(* Logix 5000 project; controller SEER_TEMPLATE vendor 1 type 14 code 54 rev 17.2; software revision 17.00 *)
// SEER_TEMPLATE

TASK MainTask (continuous, watchdog 500 ms) : MainProgram

MODULES
   Local : vendor 1 type 14 code 54 (ICP 0, rev 17.2)
END_MODULES

VAR_GLOBAL   (* controller tags *)
   F101x0 : REAL;   // SEER_IO_1 ANALOG COMM NULL REGISTER(S)
   F101x1 : REAL;   // SEER_IO_1 ANALOG COMM CYCLE TOTALIZER
   F101x2 : REAL;   // SEER_IO_1 ANALOG COMM JOB NUMBER
   F101x3 : REAL;   // SEER_IO_1 ANALOG COMM SCHEDULE NUMBER
   F101x4 : REAL;   // SEER_IO_1 ANALOG COMM OPERATOR ID
   N100x0 : INT;   // SEER_IO_0 DISCRETE COMM BINARY ELEMENTS INCLUDED
        .1   // SEER_IO_0 DISCRETE COMM CYCLE RESET COMMAND TRIGGER
        .2   // SEER_IO_0 DISCRETE COMM CYCLE RESET ONE SHOT
        .3   // SEER_IO_0 DISCRETE COMM MACHINE IS IN MAINTENANCE MODE
        .4   // SEER_IO_0 DISCRETE COMM CYCLE COUNT +1 ONE SHOT
        .5   // SEER_IO_0 DISCRETE COMM CYCLE COUNT +1 CYCLE DETECTED
        .6   // SEER_IO_0 DISCRETE COMM NO MACHINE ALARMS HAVE BEEN DETECTED
        .7   // SEER_IO_0 DISCRETE COMM NO MAJOR ALARMS HAVE BEEN DETECTED
        .8   // SEER_IO_0 DISCRETE COMM NO MINOR ALARMS HAVE BEEN DETECTED
        .9   // SEER_IO_0 DISCRETE COMM IDLE WITHOUT CYCLE DETECTED
        .11   // SEER_IO_0 DISCRETE COMM JOB '0' ONE SHOT
        .12   // SEER_IO_0 DISCRETE COMM JOB '0' ACTIVE NO JOB RUNNING
        .10   // SEER_IO_0 DISCRETE COMM ALWAYS FALSE INSTRUCTION (ALWAYS = 0)
   N100x1 : INT;   // SEER_IO_0 TEMPLATE TUTORIAL REGISTERS (REPLACE WITH YOUR BITS AND TAGS)
        .0   // SEER_IO_0 TEMPLATE TUTORIAL REPLACE WITH SOME LOGIC TO INDICATE PACKAGE TYPE "1"
        .1   // SEER_IO_0 TEMPLATE TUTORIAL REPLACE WITH SOME LOGIC TO INDICATE PACKAGE TYPE "2"
        .2   // SEER_IO_0 TEMPLATE TUTORIAL REPLACE WITH SOME LOGIC TO INDICATE PACKAGE TYPE "3"
        .3   // SEER_IO_0 TEMPLATE TUTORIAL REPLACE WITH SOME LOGIC TO INDICATE CUSTOM ALARM "1"
        .4   // SEER_IO_0 TEMPLATE TUTORIAL REPLACE WITH SOME LOGIC TO INDICATE CUSTOM ALARM "2"
        .5   // SEER_IO_0 TEMPLATE TUTORIAL REPLACE WITH SOME LOGIC TO INDICATE CUSTOM ALARM "3"
        .6   // SEER_IO_0 TEMPLATE TUTORIAL REPLACE WITH SOME LOGIC TO INDICATE CUSTOM ALARM "4"
        .7   // SEER_IO_0 TEMPLATE TUTORIAL REPLACE WITH SOME LOGIC TO INDICATE CUSTOM WARNING "1"
        .8   // SEER_IO_0 TEMPLATE TUTORIAL REPLACE WITH SOME LOGIC TO INDICATE CUSTOM WARNING "2"
        .9   // SEER_IO_0 TEMPLATE TUTORIAL REPLACE WITH SOME LOGIC TO INDICATE CUSTOM WARNING "3"
        .10   // SEER_IO_0 TEMPLATE TUTORIAL REPLACE WITH SOME LOGIC TO INDICATE THAT THE MACHINE HAS CYCLED 1 TIME
   N100x2 : INT;   // SEER_IO_0 DISCRETE COMM ALARM STATE
   N100x3 : INT;   // SEER_IO_0 DISCRETE COMM ALARM STATE PENDING
   N100x4 : INT;   // SEER_IO_0 DISCRETE COMM MACHINE STATE
   N100x5 : INT;   // SEER_IO_0 DISCRETE COMM CORRECTIVE ACTION
   N100x6 : INT;   // SEER_IO_0 DISCRETE COMM PACKAGES PER CYCLE
   N100x7 : INT;   // SEER_IO_0 DISCRETE COMM PACKAGE CLASS (TYPE)
   N100x8 : INT;   // SEER_IO_0 DISCRETE COMM MAJOR ALARM ID PENDING
   N100x9 : INT;   // SEER_IO_0 DISCRETE COMM MINOR ALARM ID PENDING
   T102x0 : TIMER := (PRE := 240000);   // SEER_IO_2 TIMERS IDLE TIME WITHOUT CYCLE DETECTED TIME BASE = 0.001 SEC
END_VAR

PROGRAM MainProgram   (* main routine MainRoutine *)

ROUTINE MainRoutine   (* ladder *)
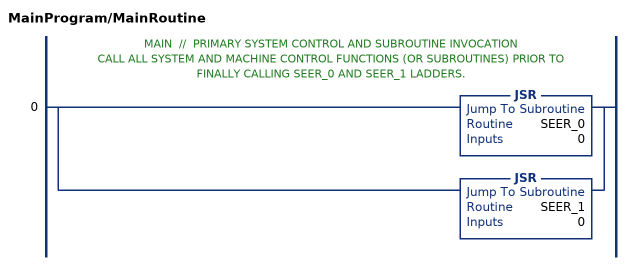
   // MAIN  //  PRIMARY SYSTEM CONTROL AND SUBROUTINE INVOCATION
   // CALL ALL SYSTEM AND MACHINE CONTROL FUNCTIONS (OR SUBROUTINES) PRIOR TO
   // FINALLY CALLING SEER_0 AND SEER_1 LADDERS.
   0: [JSR(SEER_0,0) ,JSR(SEER_1,0) ];
END_ROUTINE

ROUTINE SEER_0   (* ladder *)
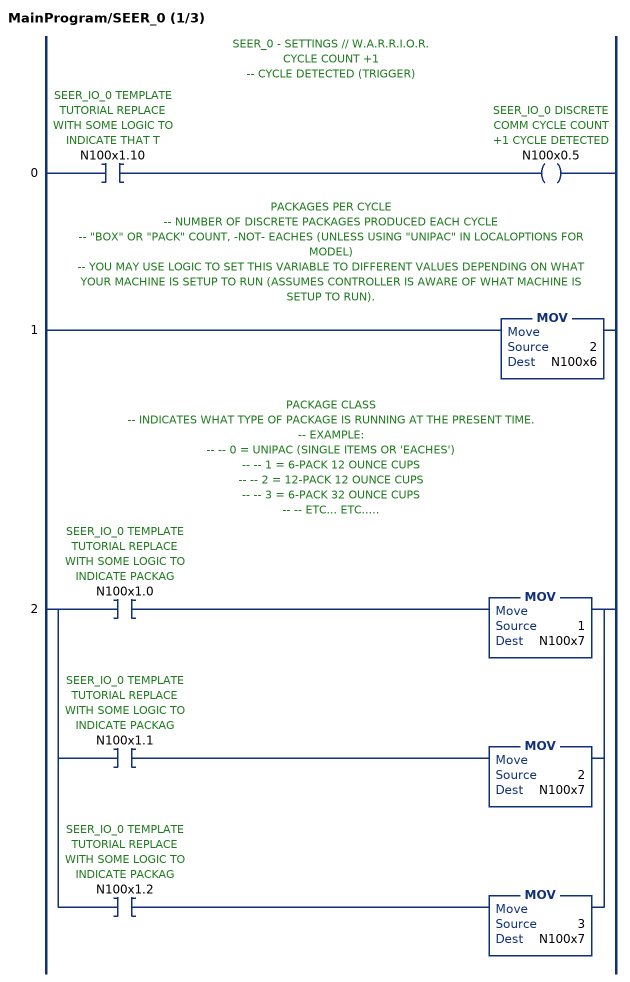
   // SEER_0 - SETTINGS // W.A.R.R.I.O.R.
   // CYCLE COUNT +1
   // -- CYCLE DETECTED (TRIGGER)
   0: XIC(N100x1.10)OTE(N100x0.5);
   // PACKAGES PER CYCLE
   // -- NUMBER OF DISCRETE PACKAGES PRODUCED EACH CYCLE
   // -- "BOX" OR "PACK" COUNT, -NOT- EACHES (UNLESS USING "UNIPAC" IN LOCALOPTIONS FOR MODEL)
   // -- YOU MAY USE LOGIC TO SET THIS VARIABLE TO DIFFERENT VALUES DEPENDING ON WHAT
   //    YOUR MACHINE IS SETUP TO RUN (ASSUMES CONTROLLER IS AWARE OF WHAT MACHINE IS
   //    SETUP TO RUN).
   1: MOV(2,N100x6);
   // PACKAGE CLASS
   // -- INDICATES WHAT TYPE OF PACKAGE IS RUNNING AT THE PRESENT TIME.
   // -- EXAMPLE:
   // -- -- 0 = UNIPAC (SINGLE ITEMS OR 'EACHES')
   // -- -- 1 = 6-PACK 12 OUNCE CUPS
   // -- -- 2 = 12-PACK 12 OUNCE CUPS
   // -- -- 3 = 6-PACK 32 OUNCE CUPS
   // -- -- ETC... ETC...
   // -- YOU MAY USE LOGIC TO SET THIS VARIABLE TO DIFFERENT VALUES DEPENDING ON WHAT
   //    YOUR MACHINE IS SETUP TO RUN (ASSUMES CONTROLLER IS AWARE OF WHAT MACHINE IS
   //    SETUP TO RUN).
   2: [XIC(N100x1.0) MOV(1,N100x7) ,XIC(N100x1.1) MOV(2,N100x7) ,XIC(N100x1.2) MOV(3,N100x7) ];
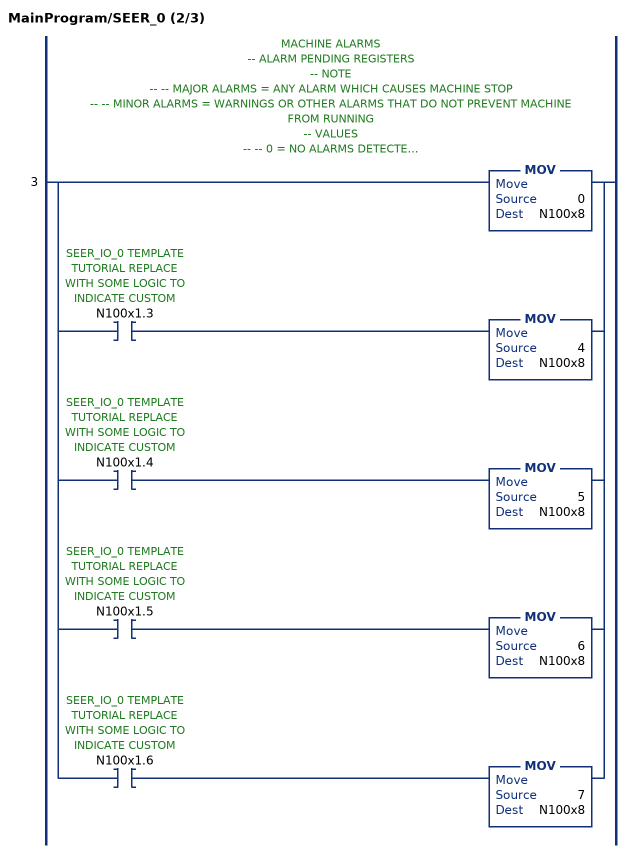
   // MACHINE ALARMS
   // -- ALARM PENDING REGISTERS
   // -- NOTE
   // -- -- MAJOR ALARMS = ANY ALARM WHICH CAUSES MACHINE STOP
   // -- -- MINOR ALARMS = WARNINGS OR OTHER ALARMS THAT DO NOT PREVENT MACHINE FROM RUNNING
   // -- VALUES
   // -- -- 0 = NO ALARMS DETECTED
   // -- -- 1 = MAINTENANCE MODE ENABLED
   // -- -- 2 = RESERVED - DO NOT USE
   // -- -- 3 = RESERVED - DO NOT USE
   // -- -- 4 .. ---> .. N = YOUR CUSTOM ALARMS
   3: [MOV(0,N100x8) ,XIC(N100x1.3) MOV(4,N100x8) ,XIC(N100x1.4) MOV(5,N100x8) ,XIC(N100x1.5) MOV(6,N100x8) ,XIC(N100x1.6) MOV(7,N100x8) ];
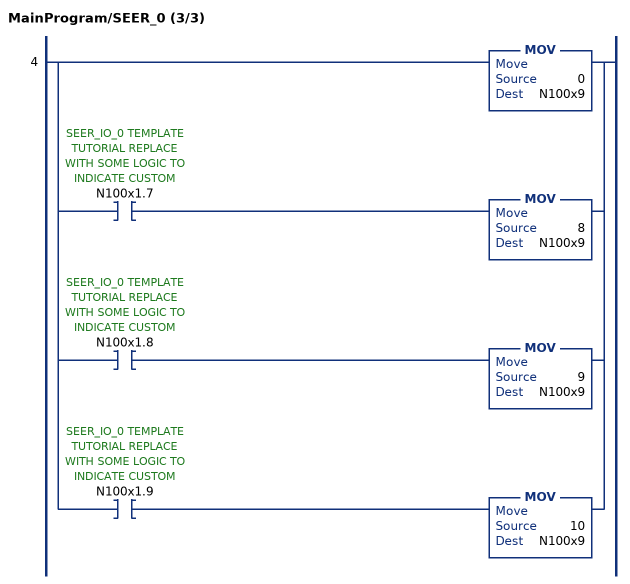
   4: [MOV(0,N100x9) ,XIC(N100x1.7) MOV(8,N100x9) ,XIC(N100x1.8) MOV(9,N100x9) ,XIC(N100x1.9) MOV(10,N100x9) ];
END_ROUTINE

ROUTINE SEER_1   (* ladder *)
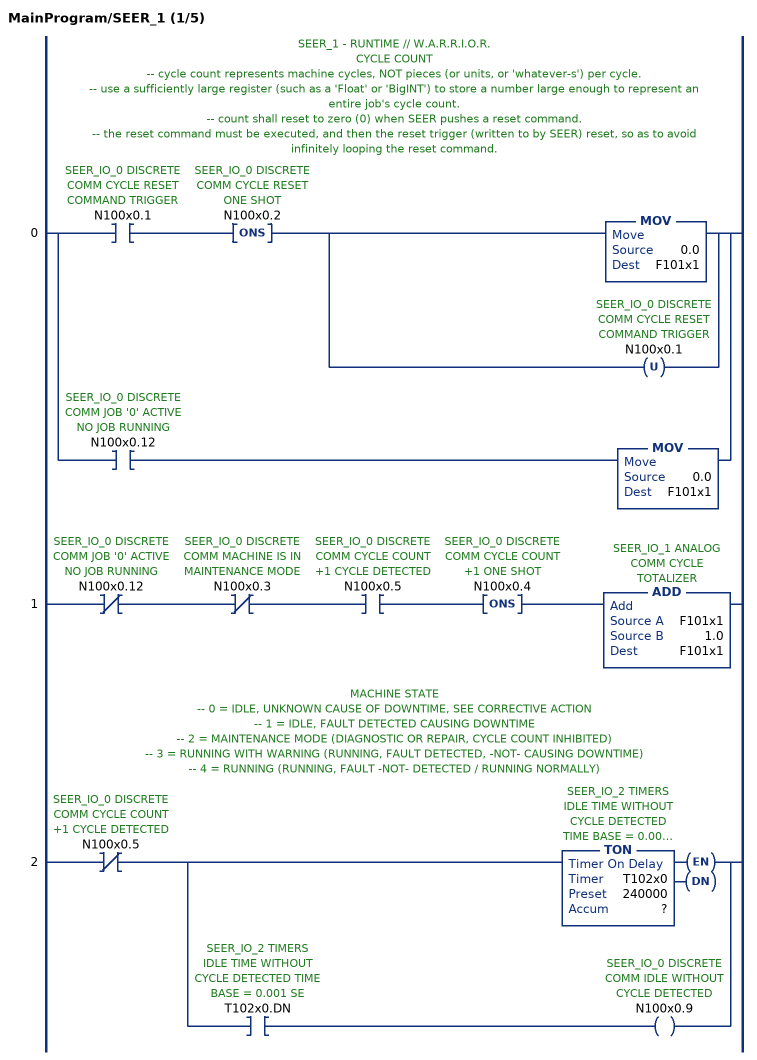
   // SEER_1 - RUNTIME // W.A.R.R.I.O.R.
   // CYCLE COUNT
   // -- cycle count represents machine cycles, NOT pieces (or units, or 'whatever-s') per cycle.
   // -- use a sufficiently large register (such as a 'Float' or 'BigINT') to store a number large enough to represent an entire job's cycle count.
   // -- count shall reset to zero (0) when SEER pushes a reset command.
   // -- the reset command must be executed, and then the reset trigger (written to by SEER) reset, so as to avoid infinitely looping the reset command.
   0: [XIC(N100x0.1) ONS(N100x0.2) [MOV(0.0,F101x1) ,OTU(N100x0.1) ] ,XIC(N100x0.12) MOV(0.0,F101x1) ];
   1: XIO(N100x0.12)XIO(N100x0.3)XIC(N100x0.5)ONS(N100x0.4)ADD(F101x1,1.0,F101x1);
   // MACHINE STATE
   // -- 0 = IDLE, UNKNOWN CAUSE OF DOWNTIME, SEE CORRECTIVE ACTION
   // -- 1 = IDLE, FAULT DETECTED CAUSING DOWNTIME
   // -- 2 = MAINTENANCE MODE (DIAGNOSTIC OR REPAIR, CYCLE COUNT INHIBITED)
   // -- 3 = RUNNING WITH WARNING (RUNNING, FAULT DETECTED, -NOT- CAUSING DOWNTIME)
   // -- 4 = RUNNING (RUNNING, FAULT -NOT- DETECTED / RUNNING NORMALLY)
   2: XIO(N100x0.5)[TON(T102x0,?,?) ,XIC(T102x0.DN) OTE(N100x0.9) ];
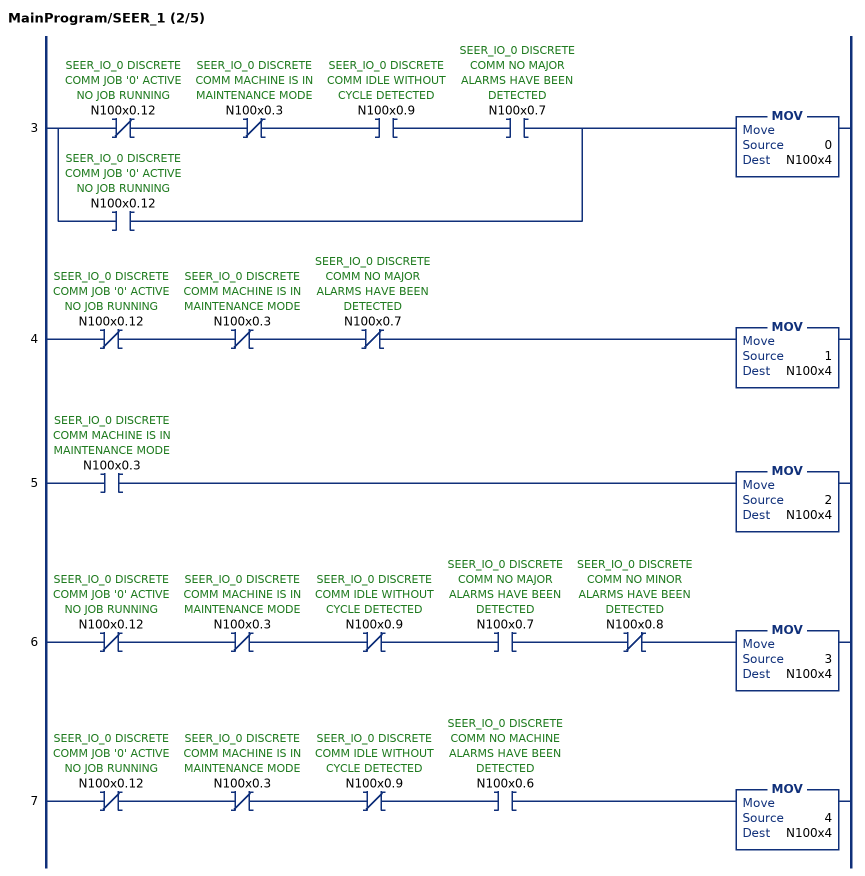
   3: [XIO(N100x0.12) XIO(N100x0.3) XIC(N100x0.9) XIC(N100x0.7) ,XIC(N100x0.12) ]MOV(0,N100x4);
   4: XIO(N100x0.12)XIO(N100x0.3)XIO(N100x0.7)MOV(1,N100x4);
   5: XIC(N100x0.3)MOV(2,N100x4);
   6: XIO(N100x0.12)XIO(N100x0.3)XIO(N100x0.9)XIC(N100x0.7)XIO(N100x0.8)MOV(3,N100x4);
   7: XIO(N100x0.12)XIO(N100x0.3)XIO(N100x0.9)XIC(N100x0.6)MOV(4,N100x4);
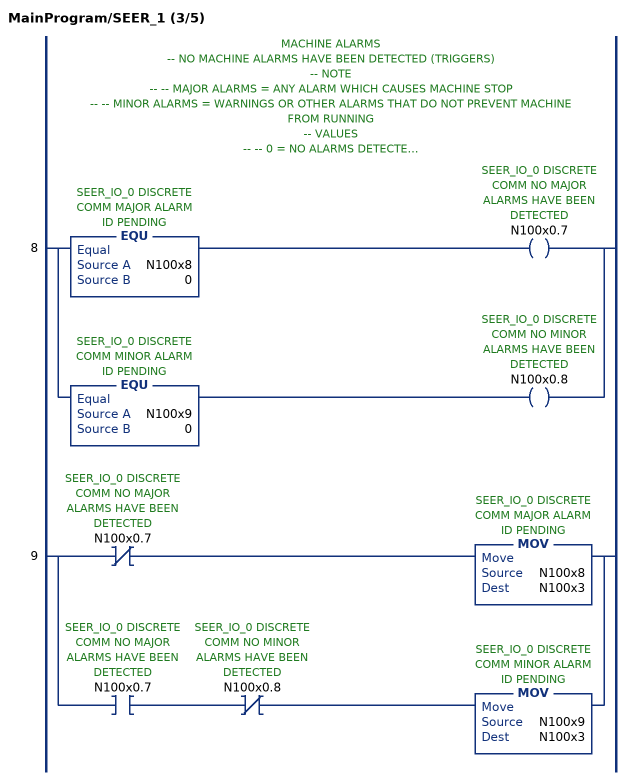
   // MACHINE ALARMS
   // -- NO MACHINE ALARMS HAVE BEEN DETECTED (TRIGGERS)
   // -- NOTE
   // -- -- MAJOR ALARMS = ANY ALARM WHICH CAUSES MACHINE STOP
   // -- -- MINOR ALARMS = WARNINGS OR OTHER ALARMS THAT DO NOT PREVENT MACHINE FROM RUNNING
   // -- VALUES
   // -- -- 0 = NO ALARMS DETECTED
   // -- -- 1 = MAINTENANCE MODE ENABLED
   // -- -- 2 = RESERVED - DO NOT USE
   // -- -- 3 = RESERVED - DO NOT USE
   // -- -- 4 .. ---> .. N = YOUR CUSTOM ALARMS
   8: [EQU(N100x8,0) OTE(N100x0.7) ,EQU(N100x9,0) OTE(N100x0.8) ];
   9: [XIO(N100x0.7) MOV(N100x8,N100x3) ,XIC(N100x0.7) XIO(N100x0.8) MOV(N100x9,N100x3) ];
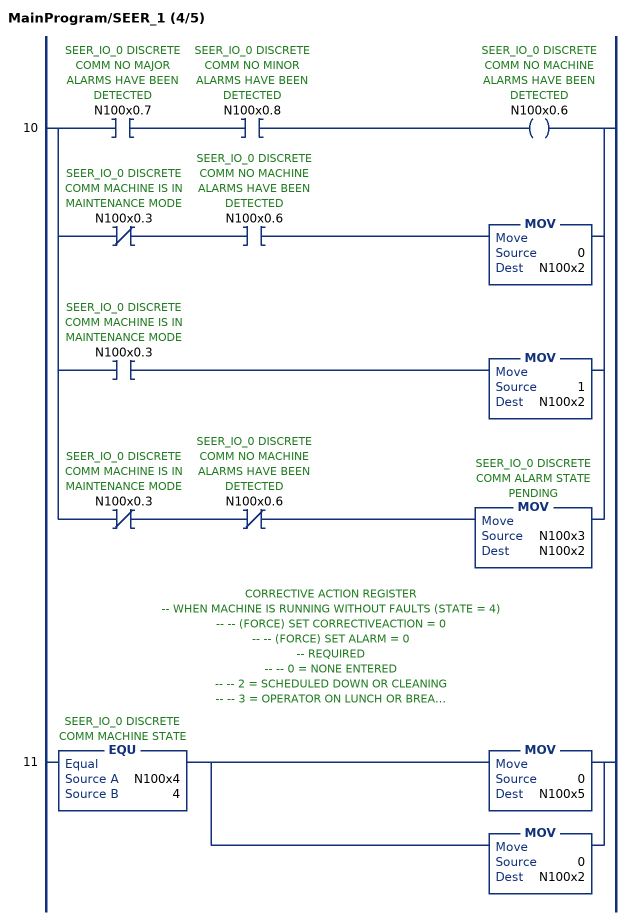
   10: [XIC(N100x0.7) XIC(N100x0.8) OTE(N100x0.6) ,XIO(N100x0.3) XIC(N100x0.6) MOV(0,N100x2) ,XIC(N100x0.3) MOV(1,N100x2) ,XIO(N100x0.3) XIO(N100x0.6) MOV(N100x3,N100x2) ];
   // CORRECTIVE ACTION REGISTER
   // -- WHEN MACHINE IS RUNNING WITHOUT FAULTS (STATE = 4)
   // -- -- (FORCE) SET CORRECTIVEACTION = 0
   // -- -- (FORCE) SET ALARM = 0
   // -- REQUIRED
   // -- -- 0 = NONE ENTERED
   // -- -- 2 = SCHEDULED DOWN OR CLEANING
   // -- -- 3 = OPERATOR ON LUNCH OR BREAK
   // -- NOTE
   // -- -- 1 DOES NOT EXIST - DEPRECATED AFTER INITIAL DEPLOYMENT
   // -- -- 2 AND 3 ARE SET BY SEER, NOT BY THE LOCAL CONTROLLER
   11: EQU(N100x4,4)[MOV(0,N100x5) ,MOV(0,N100x2) ];
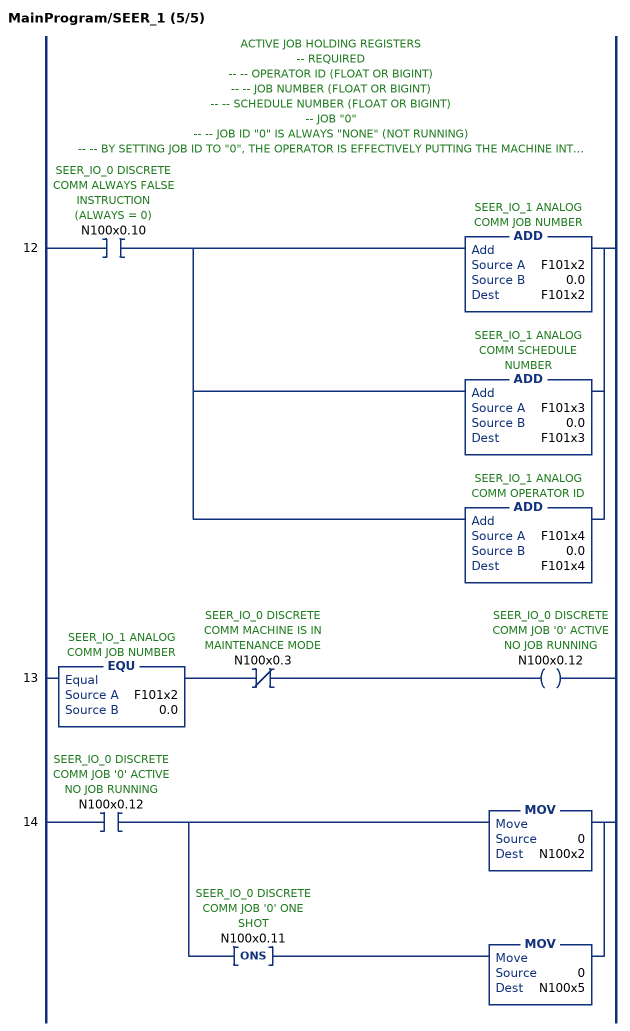
   // ACTIVE JOB HOLDING REGISTERS
   // -- REQUIRED
   // -- -- OPERATOR ID (FLOAT OR BIGINT)
   // -- -- JOB NUMBER (FLOAT OR BIGINT)
   // -- -- SCHEDULE NUMBER (FLOAT OR BIGINT)
   // -- JOB "0"
   // -- -- JOB ID "0" IS ALWAYS "NONE" (NOT RUNNING)
   // -- -- BY SETTING JOB ID TO "0", THE OPERATOR IS EFFECTIVELY PUTTING THE MACHINE INTO
   //        A FORCED "SCHEDULED DOWN OR CLEANING" ACTION, SO LET'S FORCE THAT.
   // -- NOTES
   // -- -- DO -NOT- EXECUTE LOGIC UPON THESE REGISTERS, THEY EXIST
   //        PURELY FOR USE BY SEER, WHICH WILL WRITE AND READ BACK
   //        DATA AS NEEDED.
   // -- -- THE 'ALWAYS FALSE' BIT IN FRONT OF THIS RUNG RENDERS
   //        THIS LADDER AS NOTHING MORE THAN A PLACEHOLDER FOR
   //        YOUR REFERENCE.
   12: XIC(N100x0.10)[ADD(F101x2,0.0,F101x2) ,ADD(F101x3,0.0,F101x3) ,ADD(F101x4,0.0,F101x4) ];
   13: EQU(F101x2,0.0)XIO(N100x0.3)OTE(N100x0.12);
   14: XIC(N100x0.12)[MOV(0,N100x2) ,ONS(N100x0.11) MOV(0,N100x5) ];
END_ROUTINE
END_PROGRAM
